# EPICS alarm handler configuration: mps_database/bare/alarms/areas/mpln_spd_mp04.alhConfig
GROUP NULL MPLN:SPD:MP04:1
$ALIAS MPS Link Node 95
$GUIDANCE
LTUH MPS
   Group Name: MPLN:SPD:MP04:1
   Summary PV:  MPLN:SPD:MP04:1:STATSUMY
$END
CHANNEL  MPLN:SPD:MP04:1    MPLN:SPD:MP04:1:MPS_EN_RBV		-----
CHANNEL  MPLN:SPD:MP04:1    MPLN:SPD:MP04:1:LC1_MODE_RBV		-----
